// SIMATIC STEP 7 (V5.x) project PUERTA DB
// CPU: CPU313 C-2 DP(1)
// station: P_ADR_BUS
// station: Hardware
// station: Equipo SIMATIC 300

SYMBOL_TABLE
"BIT"	DB 1	DB 1
"CONTADOR"	FB 201	FB 201	// CONTADOR CON DIFERENCIA DE OPERANDOS
"INTERMITENCIA"	FB 202	FB 202	// INTERMITENCIA CONFIGURABLE
"INGIRO"	FB 203	FB 203	// INVERSION DE GIRO
"DETECTOR"	I 0.0	BOOL
"CELULA"	I 0.1	BOOL
"FC ARRIBA"	I 0.2	BOOL
"FC ABAJO"	I 0.3	BOOL
"Cycle Execution"	OB 1	OB 1
"SUBIR"	Q 0.0	BOOL
"BAJAR"	Q 0.1	BOOL
END_SYMBOL_TABLE
